// TIA Portal V15.1 export
// export: Created 2024-06-21T08:41:01.3806409Z, ExportSetting WithDefaults, DisplayName Totally Integrated Automation Portal, DisplayVersion V15.1 Update 5, DisplayName TIA Portal Openness, DisplayVersion V15.1 Update 5, DisplayName SINAMICS Startdrive Advanced, DisplayVersion V15.1, DisplayName G130, G150, S120, S150, SINAMICS MV, S210, DisplayVersion V15.1, DisplayName G110M, G120, G120C, G120D, G120P, DisplayVersion V15.1, DisplayName STEP 7 Professional, DisplayVersion V15.1 Update 5, DisplayName STEP 7 Safety, DisplayVersion V15.1, DisplayName WinCC Professional, DisplayVersion V15.1 Update 5, DisplayName SIMATIC Visualization Architect, DisplayVersion V15.1
FUNCTION_BLOCK "LModeSummary"   // FB1004, FBD
TITLE = LModeSummary
{ S7_Optimized_Access := 'TRUE' }
AUTHOR : CSTAAL
VERSION : 0.1
// Summary of different modes
// stored: AutoNumber false, IsIECCheckEnabled false, IsRetainMemResEnabled false, MemoryReserve 100, SetENOAutomatically False, UDAEnableTagReadback false
   VAR_OUTPUT
      O_SumAutoMode { ExternalAccessible := 'False'; ExternalVisible := 'False'; ExternalWritable := 'False'} : Bool;   // Summary of Auto Mode
      O_SumAutoModeSel { ExternalAccessible := 'False'; ExternalVisible := 'False'; ExternalWritable := 'False'} : Bool;   // Summary of Auto Mode Select
      O_SumStepMode { ExternalAccessible := 'False'; ExternalVisible := 'False'; ExternalWritable := 'False'} : Bool;   // Summary of Step Mode
      O_SumStepModeSel { ExternalAccessible := 'False'; ExternalVisible := 'False'; ExternalWritable := 'False'} : Bool;   // Summary of Step Mode Select
      O_SumHomeRunMode { ExternalAccessible := 'False'; ExternalVisible := 'False'; ExternalWritable := 'False'} : Bool;   // Summary of Home Run Mode
      O_SumHomeRunModeSel { ExternalAccessible := 'False'; ExternalVisible := 'False'; ExternalWritable := 'False'} : Bool;   // Summary of Home Run Mode Secect
      O_SumManualMode { ExternalAccessible := 'False'; ExternalVisible := 'False'; ExternalWritable := 'False'} : Bool;   // Summary of Manual Mode
      O_SumManualModeSel { ExternalAccessible := 'False'; ExternalVisible := 'False'; ExternalWritable := 'False'} : Bool;   // Summary of Manual Mode Select
      O_SumAnyProdModeActive { ExternalAccessible := 'False'; ExternalVisible := 'False'; ExternalWritable := 'False'} : Bool;   // Summary of Any Production Mode Active
      O_SumAnyProdModeSel { ExternalAccessible := 'False'; ExternalVisible := 'False'; ExternalWritable := 'False'} : Bool;   // Summary of Any Production Mode Select
      O_SumMode { ExternalAccessible := 'False'; ExternalVisible := 'False'; ExternalWritable := 'False'} : "Modes";   // Summary Mode
   END_VAR
   VAR_IN_OUT
      IO_ModesZM1 : "Modes";   // Modes ZM1
      IO_ModesZM2 : "Modes";   // Modes ZM2
      IO_ModesZM3 : "Modes";   // Modes ZM3
      IO_ModesZM4 : "Modes";   // Modes ZM4
      IO_ModesZM5 : "Modes";   // Modes ZM5
   END_VAR
BEGIN

REGION Network 1: **** 8 - Outputs **** Summary Auto Mode
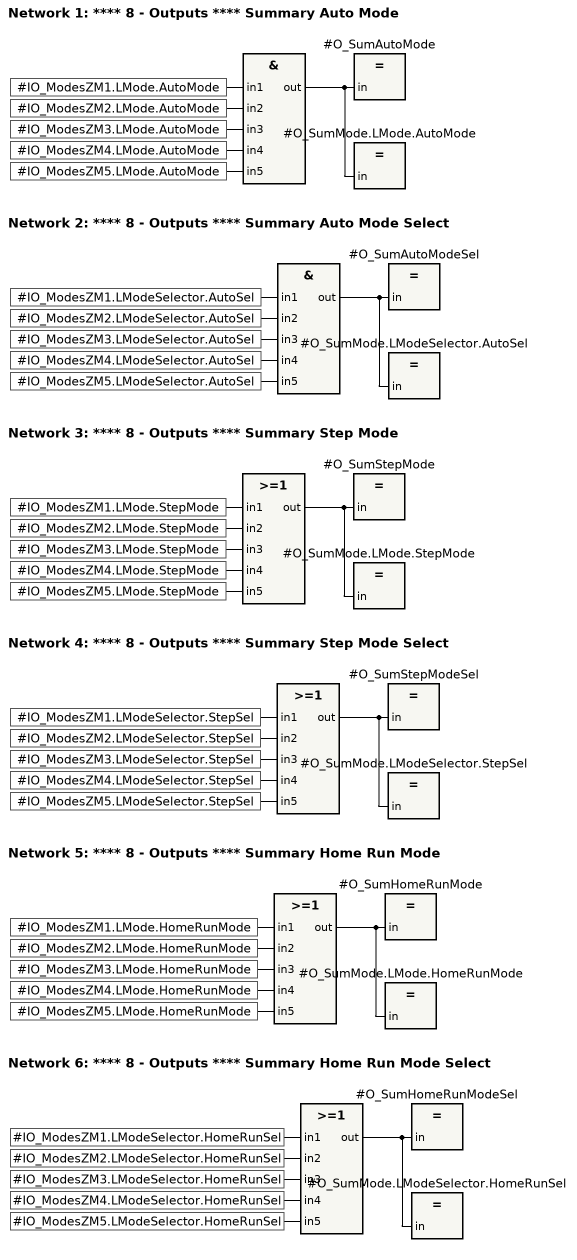
   #O_SumAutoMode := #IO_ModesZM1.LMode.AutoMode AND #IO_ModesZM2.LMode.AutoMode AND #IO_ModesZM3.LMode.AutoMode AND #IO_ModesZM4.LMode.AutoMode AND #IO_ModesZM5.LMode.AutoMode;
   #O_SumMode.LMode.AutoMode := #O_SumAutoMode;
END_REGION

REGION Network 2: **** 8 - Outputs **** Summary Auto Mode Select
   #O_SumAutoModeSel := #IO_ModesZM1.LModeSelector.AutoSel AND #IO_ModesZM2.LModeSelector.AutoSel AND #IO_ModesZM3.LModeSelector.AutoSel AND #IO_ModesZM4.LModeSelector.AutoSel AND #IO_ModesZM5.LModeSelector.AutoSel;
   #O_SumMode.LModeSelector.AutoSel := #O_SumAutoModeSel;
END_REGION

REGION Network 3: **** 8 - Outputs **** Summary Step Mode
   #O_SumStepMode := #IO_ModesZM1.LMode.StepMode OR #IO_ModesZM2.LMode.StepMode OR #IO_ModesZM3.LMode.StepMode OR #IO_ModesZM4.LMode.StepMode OR #IO_ModesZM5.LMode.StepMode;
   #O_SumMode.LMode.StepMode := #O_SumStepMode;
END_REGION

REGION Network 4: **** 8 - Outputs **** Summary Step Mode Select
   #O_SumStepModeSel := #IO_ModesZM1.LModeSelector.StepSel OR #IO_ModesZM2.LModeSelector.StepSel OR #IO_ModesZM3.LModeSelector.StepSel OR #IO_ModesZM4.LModeSelector.StepSel OR #IO_ModesZM5.LModeSelector.StepSel;
   #O_SumMode.LModeSelector.StepSel := #O_SumStepModeSel;
END_REGION

REGION Network 5: **** 8 - Outputs **** Summary Home Run Mode
   #O_SumHomeRunMode := #IO_ModesZM1.LMode.HomeRunMode OR #IO_ModesZM2.LMode.HomeRunMode OR #IO_ModesZM3.LMode.HomeRunMode OR #IO_ModesZM4.LMode.HomeRunMode OR #IO_ModesZM5.LMode.HomeRunMode;
   #O_SumMode.LMode.HomeRunMode := #O_SumHomeRunMode;
END_REGION

REGION Network 6: **** 8 - Outputs **** Summary Home Run Mode Select
   #O_SumHomeRunModeSel := #IO_ModesZM1.LModeSelector.HomeRunSel OR #IO_ModesZM2.LModeSelector.HomeRunSel OR #IO_ModesZM3.LModeSelector.HomeRunSel OR #IO_ModesZM4.LModeSelector.HomeRunSel OR #IO_ModesZM5.LModeSelector.HomeRunSel;
   #O_SumMode.LModeSelector.HomeRunSel := #O_SumHomeRunModeSel;
END_REGION

REGION Network 7: **** 8 - Outputs **** Summary Manual Mode
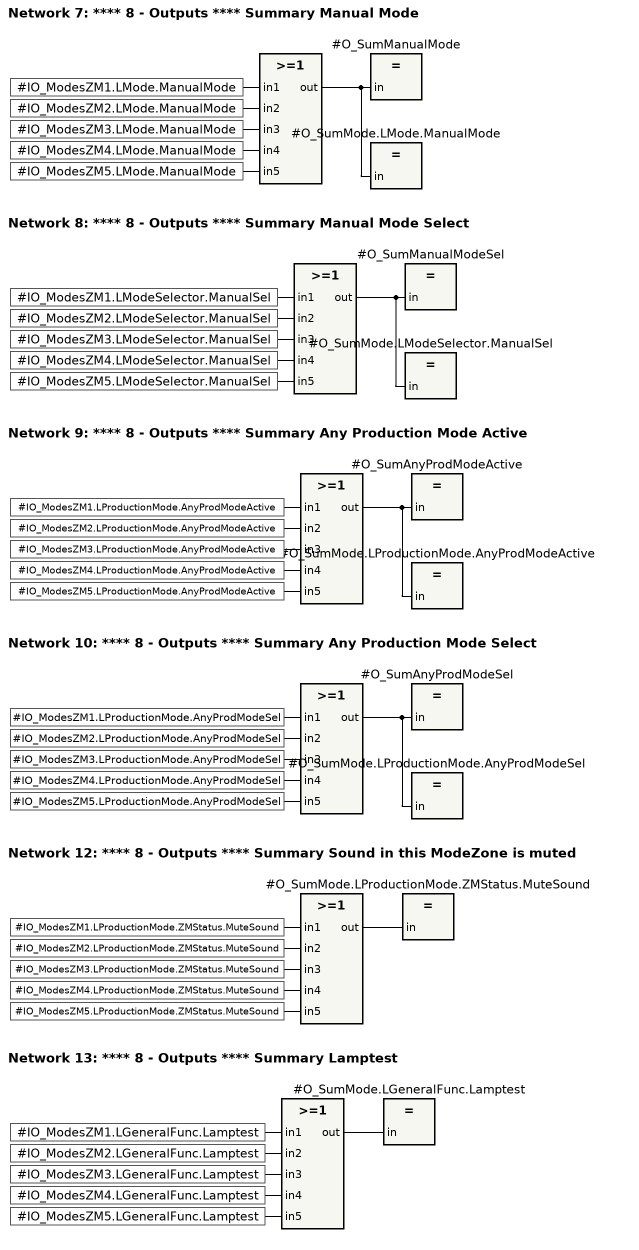
   #O_SumManualMode := #IO_ModesZM1.LMode.ManualMode OR #IO_ModesZM2.LMode.ManualMode OR #IO_ModesZM3.LMode.ManualMode OR #IO_ModesZM4.LMode.ManualMode OR #IO_ModesZM5.LMode.ManualMode;
   #O_SumMode.LMode.ManualMode := #O_SumManualMode;
END_REGION

REGION Network 8: **** 8 - Outputs **** Summary Manual Mode Select
   #O_SumManualModeSel := #IO_ModesZM1.LModeSelector.ManualSel OR #IO_ModesZM2.LModeSelector.ManualSel OR #IO_ModesZM3.LModeSelector.ManualSel OR #IO_ModesZM4.LModeSelector.ManualSel OR #IO_ModesZM5.LModeSelector.ManualSel;
   #O_SumMode.LModeSelector.ManualSel := #O_SumManualModeSel;
END_REGION

REGION Network 9: **** 8 - Outputs **** Summary Any Production Mode Active
   #O_SumAnyProdModeActive := #IO_ModesZM1.LProductionMode.AnyProdModeActive OR #IO_ModesZM2.LProductionMode.AnyProdModeActive OR #IO_ModesZM3.LProductionMode.AnyProdModeActive OR #IO_ModesZM4.LProductionMode.AnyProdModeActive OR #IO_ModesZM5.LProductionMode.AnyProdModeActive;
   #O_SumMode.LProductionMode.AnyProdModeActive := #O_SumAnyProdModeActive;
END_REGION

REGION Network 10: **** 8 - Outputs **** Summary Any Production Mode Select
   #O_SumAnyProdModeSel := #IO_ModesZM1.LProductionMode.AnyProdModeSel OR #IO_ModesZM2.LProductionMode.AnyProdModeSel OR #IO_ModesZM3.LProductionMode.AnyProdModeSel OR #IO_ModesZM4.LProductionMode.AnyProdModeSel OR #IO_ModesZM5.LProductionMode.AnyProdModeSel;
   #O_SumMode.LProductionMode.AnyProdModeSel := #O_SumAnyProdModeSel;
END_REGION

REGION Network 11: **** --------------------- Extra --------------------- ****
END_REGION

REGION Network 12: **** 8 - Outputs **** Summary Sound in this ModeZone is muted
   #O_SumMode.LProductionMode.ZMStatus.MuteSound := #IO_ModesZM1.LProductionMode.ZMStatus.MuteSound OR #IO_ModesZM2.LProductionMode.ZMStatus.MuteSound OR #IO_ModesZM3.LProductionMode.ZMStatus.MuteSound OR #IO_ModesZM4.LProductionMode.ZMStatus.MuteSound OR #IO_ModesZM5.LProductionMode.ZMStatus.MuteSound;
END_REGION

REGION Network 13: **** 8 - Outputs **** Summary Lamptest
   #O_SumMode.LGeneralFunc.Lamptest := #IO_ModesZM1.LGeneralFunc.Lamptest OR #IO_ModesZM2.LGeneralFunc.Lamptest OR #IO_ModesZM3.LGeneralFunc.Lamptest OR #IO_ModesZM4.LGeneralFunc.Lamptest OR #IO_ModesZM5.LGeneralFunc.Lamptest;
END_REGION

REGION Network 14: ***** 8 - Outputs **** Summary Lamptest steady
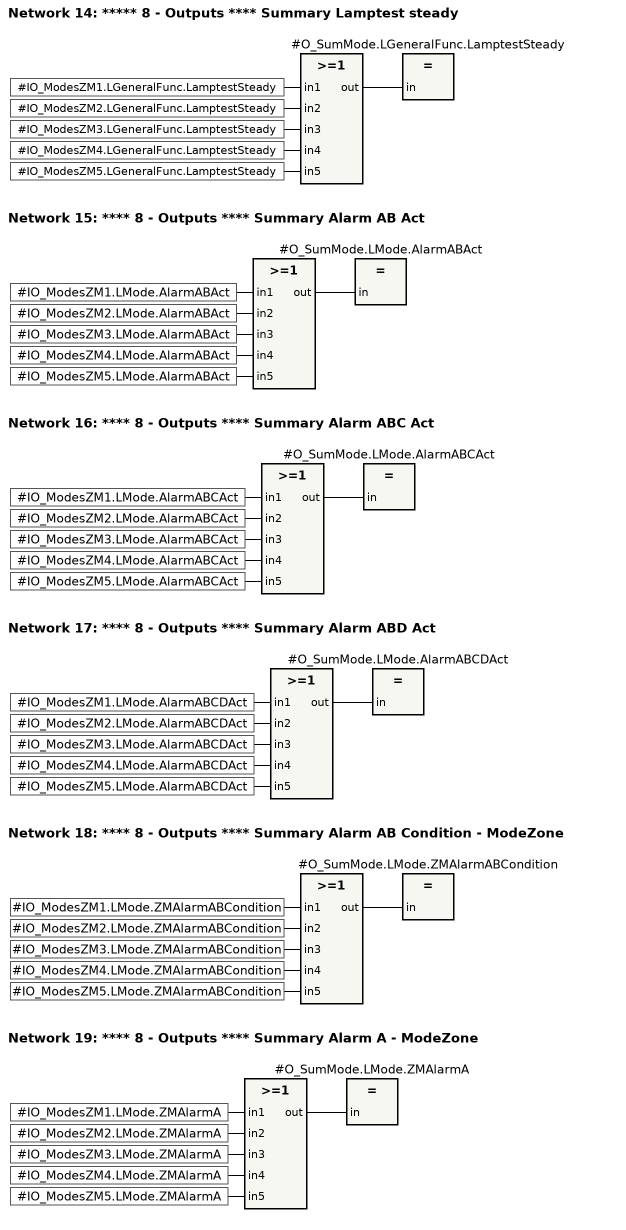
   #O_SumMode.LGeneralFunc.LamptestSteady := #IO_ModesZM1.LGeneralFunc.LamptestSteady OR #IO_ModesZM2.LGeneralFunc.LamptestSteady OR #IO_ModesZM3.LGeneralFunc.LamptestSteady OR #IO_ModesZM4.LGeneralFunc.LamptestSteady OR #IO_ModesZM5.LGeneralFunc.LamptestSteady;
END_REGION

REGION Network 15: **** 8 - Outputs **** Summary Alarm AB Act
   #O_SumMode.LMode.AlarmABAct := #IO_ModesZM1.LMode.AlarmABAct OR #IO_ModesZM2.LMode.AlarmABAct OR #IO_ModesZM3.LMode.AlarmABAct OR #IO_ModesZM4.LMode.AlarmABAct OR #IO_ModesZM5.LMode.AlarmABAct;
END_REGION

REGION Network 16: **** 8 - Outputs **** Summary Alarm ABC Act
   #O_SumMode.LMode.AlarmABCAct := #IO_ModesZM1.LMode.AlarmABCAct OR #IO_ModesZM2.LMode.AlarmABCAct OR #IO_ModesZM3.LMode.AlarmABCAct OR #IO_ModesZM4.LMode.AlarmABCAct OR #IO_ModesZM5.LMode.AlarmABCAct;
END_REGION

REGION Network 17: **** 8 - Outputs **** Summary Alarm ABD Act
   #O_SumMode.LMode.AlarmABCDAct := #IO_ModesZM1.LMode.AlarmABCDAct OR #IO_ModesZM2.LMode.AlarmABCDAct OR #IO_ModesZM3.LMode.AlarmABCDAct OR #IO_ModesZM4.LMode.AlarmABCDAct OR #IO_ModesZM5.LMode.AlarmABCDAct;
END_REGION

REGION Network 18: **** 8 - Outputs **** Summary Alarm AB Condition - ModeZone
   #O_SumMode.LMode.ZMAlarmABCondition := #IO_ModesZM1.LMode.ZMAlarmABCondition OR #IO_ModesZM2.LMode.ZMAlarmABCondition OR #IO_ModesZM3.LMode.ZMAlarmABCondition OR #IO_ModesZM4.LMode.ZMAlarmABCondition OR #IO_ModesZM5.LMode.ZMAlarmABCondition;
END_REGION

REGION Network 19: **** 8 - Outputs **** Summary Alarm A - ModeZone
   #O_SumMode.LMode.ZMAlarmA := #IO_ModesZM1.LMode.ZMAlarmA OR #IO_ModesZM2.LMode.ZMAlarmA OR #IO_ModesZM3.LMode.ZMAlarmA OR #IO_ModesZM4.LMode.ZMAlarmA OR #IO_ModesZM5.LMode.ZMAlarmA;
END_REGION

REGION Network 20: **** 8 - Outputs **** Summary Alarm B - ModeZone
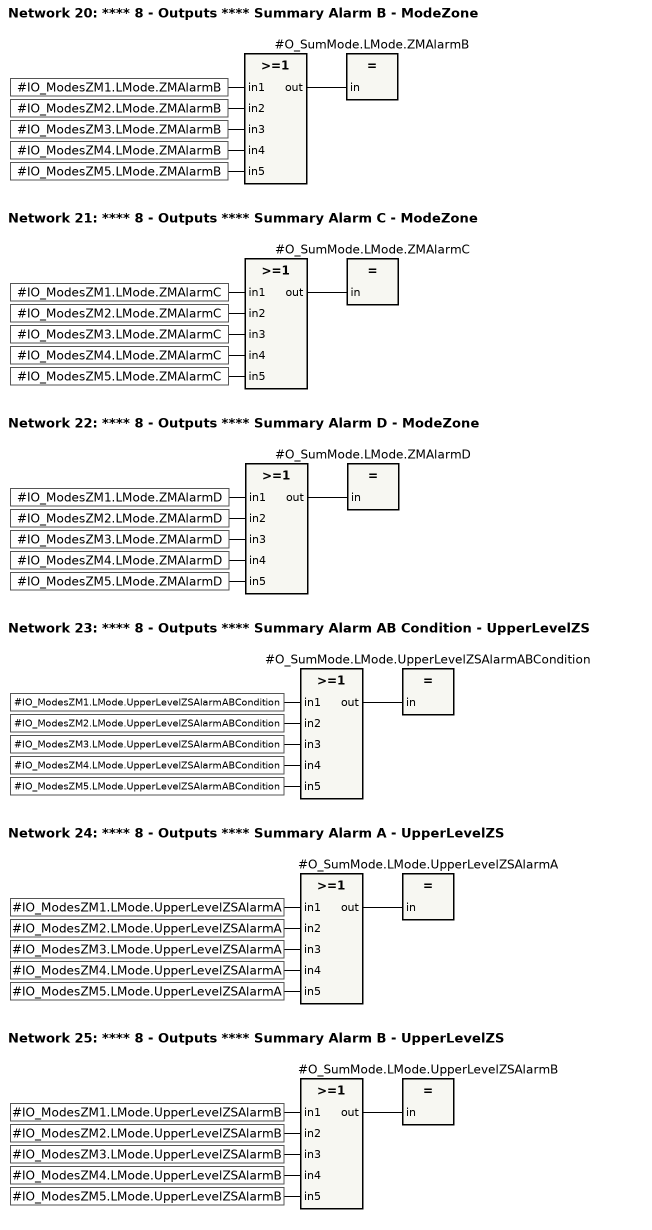
   #O_SumMode.LMode.ZMAlarmB := #IO_ModesZM1.LMode.ZMAlarmB OR #IO_ModesZM2.LMode.ZMAlarmB OR #IO_ModesZM3.LMode.ZMAlarmB OR #IO_ModesZM4.LMode.ZMAlarmB OR #IO_ModesZM5.LMode.ZMAlarmB;
END_REGION

REGION Network 21: **** 8 - Outputs **** Summary Alarm C - ModeZone
   #O_SumMode.LMode.ZMAlarmC := #IO_ModesZM1.LMode.ZMAlarmC OR #IO_ModesZM2.LMode.ZMAlarmC OR #IO_ModesZM3.LMode.ZMAlarmC OR #IO_ModesZM4.LMode.ZMAlarmC OR #IO_ModesZM5.LMode.ZMAlarmC;
END_REGION

REGION Network 22: **** 8 - Outputs **** Summary Alarm D - ModeZone
   #O_SumMode.LMode.ZMAlarmD := #IO_ModesZM1.LMode.ZMAlarmD OR #IO_ModesZM2.LMode.ZMAlarmD OR #IO_ModesZM3.LMode.ZMAlarmD OR #IO_ModesZM4.LMode.ZMAlarmD OR #IO_ModesZM5.LMode.ZMAlarmD;
END_REGION

REGION Network 23: **** 8 - Outputs **** Summary Alarm AB Condition - UpperLevelZS
   #O_SumMode.LMode.UpperLevelZSAlarmABCondition := #IO_ModesZM1.LMode.UpperLevelZSAlarmABCondition OR #IO_ModesZM2.LMode.UpperLevelZSAlarmABCondition OR #IO_ModesZM3.LMode.UpperLevelZSAlarmABCondition OR #IO_ModesZM4.LMode.UpperLevelZSAlarmABCondition OR #IO_ModesZM5.LMode.UpperLevelZSAlarmABCondition;
END_REGION

REGION Network 24: **** 8 - Outputs **** Summary Alarm A - UpperLevelZS
   #O_SumMode.LMode.UpperLevelZSAlarmA := #IO_ModesZM1.LMode.UpperLevelZSAlarmA OR #IO_ModesZM2.LMode.UpperLevelZSAlarmA OR #IO_ModesZM3.LMode.UpperLevelZSAlarmA OR #IO_ModesZM4.LMode.UpperLevelZSAlarmA OR #IO_ModesZM5.LMode.UpperLevelZSAlarmA;
END_REGION

REGION Network 25: **** 8 - Outputs **** Summary Alarm B - UpperLevelZS
   #O_SumMode.LMode.UpperLevelZSAlarmB := #IO_ModesZM1.LMode.UpperLevelZSAlarmB OR #IO_ModesZM2.LMode.UpperLevelZSAlarmB OR #IO_ModesZM3.LMode.UpperLevelZSAlarmB OR #IO_ModesZM4.LMode.UpperLevelZSAlarmB OR #IO_ModesZM5.LMode.UpperLevelZSAlarmB;
END_REGION

REGION Network 26: **** 8 - Outputs **** Summary Alarm C - UpperLevelZS
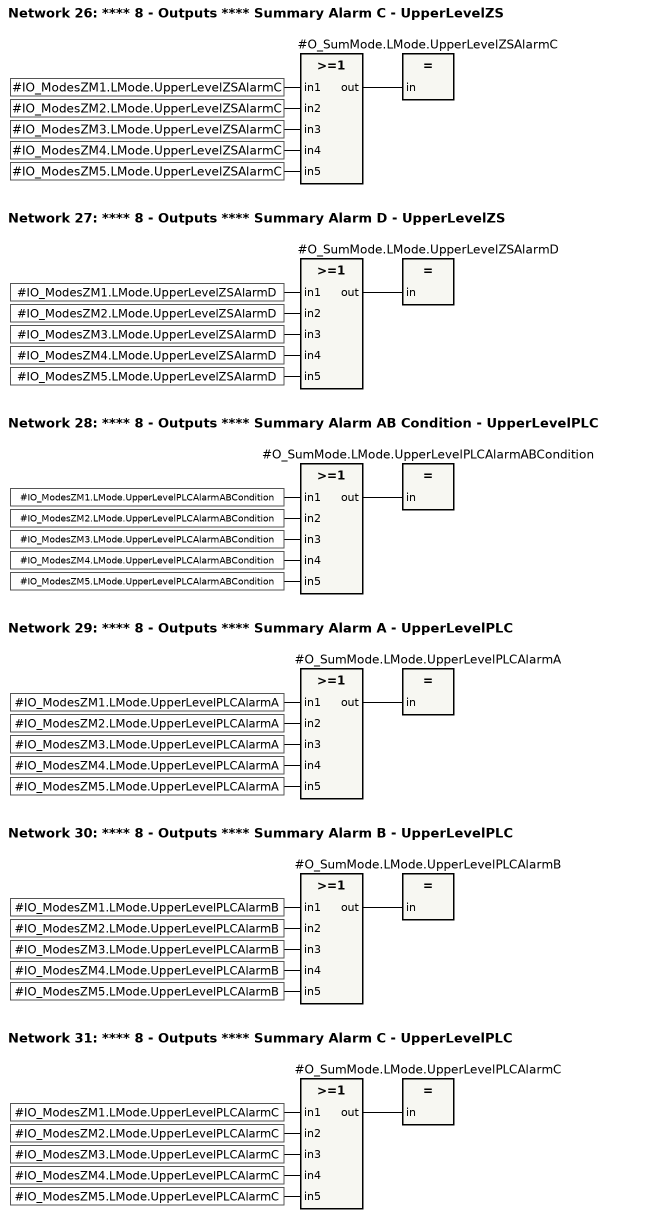
   #O_SumMode.LMode.UpperLevelZSAlarmC := #IO_ModesZM1.LMode.UpperLevelZSAlarmC OR #IO_ModesZM2.LMode.UpperLevelZSAlarmC OR #IO_ModesZM3.LMode.UpperLevelZSAlarmC OR #IO_ModesZM4.LMode.UpperLevelZSAlarmC OR #IO_ModesZM5.LMode.UpperLevelZSAlarmC;
END_REGION

REGION Network 27: **** 8 - Outputs **** Summary Alarm D - UpperLevelZS
   #O_SumMode.LMode.UpperLevelZSAlarmD := #IO_ModesZM1.LMode.UpperLevelZSAlarmD OR #IO_ModesZM2.LMode.UpperLevelZSAlarmD OR #IO_ModesZM3.LMode.UpperLevelZSAlarmD OR #IO_ModesZM4.LMode.UpperLevelZSAlarmD OR #IO_ModesZM5.LMode.UpperLevelZSAlarmD;
END_REGION

REGION Network 28: **** 8 - Outputs **** Summary Alarm AB Condition - UpperLevelPLC
   #O_SumMode.LMode.UpperLevelPLCAlarmABCondition := #IO_ModesZM1.LMode.UpperLevelPLCAlarmABCondition OR #IO_ModesZM2.LMode.UpperLevelPLCAlarmABCondition OR #IO_ModesZM3.LMode.UpperLevelPLCAlarmABCondition OR #IO_ModesZM4.LMode.UpperLevelPLCAlarmABCondition OR #IO_ModesZM5.LMode.UpperLevelPLCAlarmABCondition;
END_REGION

REGION Network 29: **** 8 - Outputs **** Summary Alarm A - UpperLevelPLC
   #O_SumMode.LMode.UpperLevelPLCAlarmA := #IO_ModesZM1.LMode.UpperLevelPLCAlarmA OR #IO_ModesZM2.LMode.UpperLevelPLCAlarmA OR #IO_ModesZM3.LMode.UpperLevelPLCAlarmA OR #IO_ModesZM4.LMode.UpperLevelPLCAlarmA OR #IO_ModesZM5.LMode.UpperLevelPLCAlarmA;
END_REGION

REGION Network 30: **** 8 - Outputs **** Summary Alarm B - UpperLevelPLC
   #O_SumMode.LMode.UpperLevelPLCAlarmB := #IO_ModesZM1.LMode.UpperLevelPLCAlarmB OR #IO_ModesZM2.LMode.UpperLevelPLCAlarmB OR #IO_ModesZM3.LMode.UpperLevelPLCAlarmB OR #IO_ModesZM4.LMode.UpperLevelPLCAlarmB OR #IO_ModesZM5.LMode.UpperLevelPLCAlarmB;
END_REGION

REGION Network 31: **** 8 - Outputs **** Summary Alarm C - UpperLevelPLC
   #O_SumMode.LMode.UpperLevelPLCAlarmC := #IO_ModesZM1.LMode.UpperLevelPLCAlarmC OR #IO_ModesZM2.LMode.UpperLevelPLCAlarmC OR #IO_ModesZM3.LMode.UpperLevelPLCAlarmC OR #IO_ModesZM4.LMode.UpperLevelPLCAlarmC OR #IO_ModesZM5.LMode.UpperLevelPLCAlarmC;
END_REGION

REGION Network 32: **** 8 - Outputs **** Summary Alarm D - UpperLevelPLC
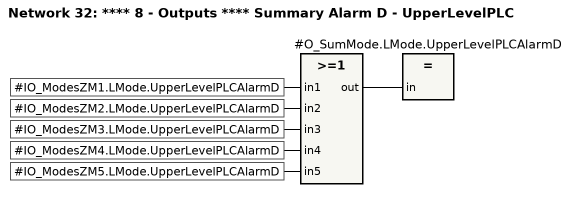
   #O_SumMode.LMode.UpperLevelPLCAlarmD := #IO_ModesZM1.LMode.UpperLevelPLCAlarmD OR #IO_ModesZM2.LMode.UpperLevelPLCAlarmD OR #IO_ModesZM3.LMode.UpperLevelPLCAlarmD OR #IO_ModesZM4.LMode.UpperLevelPLCAlarmD OR #IO_ModesZM5.LMode.UpperLevelPLCAlarmD;
END_REGION

REGION Network 33: **** -------------------------------------------------- ****
END_REGION
END_FUNCTION_BLOCK
